// TwinCAT 3 PLC project TC
// ProgramVersion: 3.1.4022.3
// libraries:
//   Tc2_Standard, * (Beckhoff Automation GmbH)
//   Tc2_System, * (Beckhoff Automation GmbH)
//   Tc2_Utilities, * (Beckhoff Automation GmbH)
//   Tc3_EventLogger, * (Beckhoff Automation GmbH)
//   Tc3_HBI_Cylinder, * (BeckHoff SG)
//   Tc3_HBI_DataLogger, * (BeckHoff SG)
//   Tc3_HBI_System, * (BeckHoff)
//   Tc3_HBI_Utilities, * (BeckHoff SG)
//   Tc3_Module, * (Beckhoff Automation GmbH)
//   VisuDialogs, * (System)
//   VisuSymbols,3.5.10.0,System
// project tree:
//   DUTs/Actuator/ DUT_Cylinder.TcDUT, DUT_Switch.TcDUT, Enum_EPT.TcDUT, Enum_ModuleEnableState.TcDUT, Enum_Presence.TcDUT
//   DUTs/AIN/ DUT_AIN.TcDUT
//   DUTs/Enum/ E_AirValve.TcDUT, E_Cmd.TcTLEO, E_DBStnLED.TcDUT, E_FacilityState.TcDUT, E_LED.TcDUT, E_Pwr.TcDUT, E_Solenoid.TcDUT, E_TstPwrStep.TcDUT, E_BackdoorState_1.TcDUT, E_ModuleID_1.TcDUT, E_ProcessState.TcDUT, E_ProcessStep.TcDUT, E_SeqSts_1.TcDUT
//   DUTs/E_Alarm/ E_AlarmID.TcDUT, E_ColAlarm.TcDUT, E_DCFACAlarm.TcDUT, E_DSAlarm.TcDUT, E_TIIAlarm.TcDUT, ST_AlarmModules.TcDUT, ST_AlarmSubmodules.TcDUT, ST_AlarmTags.TcDUT
//   DUTs/Communication/ E_EventName.TcDUT, E_ModuleID.TcDUT, E_TaskName.TcDUT, ST_Command.TcDUT, ST_Event.TcDUT, ST_EventQueue.TcDUT, ST_TACommands.TcDUT, ST_TAEvents.TcDUT
//   DUTs/ E_BackdoorState.TcDUT, ST_StepMode.TcDUT, ST_DebugStation.TcDUT, ST_TCMultilevel.TcDUT, ST_TCShuttlePOC.TcDUT, ST_TCLevel.TcDUT
//   DUTs/HMI/ ST_BypassTII.TcDUT
//   DUTs/Logging/ F_Concat5.TcPOU
//   DUTs/ModuleState/EnableDisable/ E_State.TcDUT, ST_LPState.TcDUT, ST_LPTTS_State.TcDUT, ST_TCSubModuleState.TcDUT, ST_TCSiteState.TcDUT, ST_TTS_State.TcDUT
//   DUTs/ModuleState/EPT/ E_EPT.TcDUT, ST_LPTTS_EPT.TcDUT, ST_TCUEPT.TcDUT, ST_TCSubModuleEPT.TcDUT, ST_TC_EPT.TcDUT, ST_TTS_EPT.TcDUT
//   / GlobalTextList.TcGTLO, PlcTask.TcTTO, Visualization Manager.TcVMO (not stored)
//   GVLs/ AlarmTxtList.TcTLO, BDList.TcTLO, BtnTxtList.TcTLO, CmdTxtList.TcTLO, GVL_CONSTANTS.TcGVL, GVL_EAP.TcGVL, GVL_Motor.TcGVL, GVL_Process.TcGVL, GVL_SEN_SPEC.TcGVL, GVL_TA.TcGVL, GVL_TC.TcGVL, LevelTxtList.TcTLO
//   Image/ ImageCollection.TcIPO (not stored)
//   POUs/1%29 Main/ MAIN.TcPOU (not stored)
//   POUs/2%29 DFB/Actuator/ DFB_Cylinder.TcPOU (not stored)
//   POUs/2%29 DFB/ DFB_AIN.TcPOU (not stored), DFB_Second_Pulse.TcPOU (not stored), DFB_Switch.TcPOU (not stored)
//   POUs/2) DFB/Facility/ DFB_FacilityAlarmAnlg.TcPOU, DFB_FacilityAlarm.TcPOU, DFB_FacilityAlarm_1.TcPOU
//   POUs/2%29 DFB/Facility/ DFB_FacilityAlarmBool.TcPOU (not stored)
//   POUs/2%29 DFB/Word/ FC_BitToWord.TcPOU (not stored), FC_WordToBit.TcPOU (not stored)
//   POUs/3%29 FB/1%29 Common/EAP/ ST_DCEAP.TcDUT (not stored), ST_EAP.TcDUT (not stored), ST_TBOT_TC_EAP.TcDUT (not stored), ST_TBOT_TC_SubLevelEAP.TcDUT (not stored)
//   POUs/3%29 FB/1%29 Common/FB_Alarm/ FB_Alarm.TcPOU (not stored), FB_AlarmDelay.TcPOU (not stored), FB_Delay.TcPOU (not stored)
//   POUs/3%29 FB/1%29 Common/FB_CommonFunction/ FB_AnlgSIM.TcPOU (not stored), FB_Blink.TcPOU (not stored), F_ArrayInt.TcPOU (not stored), F_ArrayStr.TcPOU (not stored), F_Concat3.TcPOU (not stored), F_GetColumnID.TcPOU (not stored), F_GetModuleID.TcPOU (not stored), F_TAParamtoStr.TcPOU (not stored)
//   POUs/3%29 FB/1%29 Common/FB_EPT/ FB_DebugStationEPTUpdate.TcPOU (not stored), FB_TCMLevelEPTUpdate.TcPOU (not stored)
//   POUs/3%29 FB/1%29 Common/FB_Logging/ FB_AlarmMonitor.TcPOU (not stored), FB_SensorMonitor.TcPOU (not stored), F_AlarmLog.TcPOU (not stored), F_SensorLog.TcPOU (not stored), Logging.TcPOU (not stored)
//   POUs/3%29 FB/1%29 Common/FB_RemoteCmdAndEvent/ CmdAndEventProcess.TcPOU (not stored), FB_CmdAndEventUpdate.TcPOU (not stored), FB_DoorOpenClose.TcPOU (not stored), FB_TCUSafeState.TcPOU (not stored), FUN_CmdToEvent.TcPOU (not stored)
//   POUs/3%29 FB/2%29 TC/ ASSIGN_COLUMN.TcPOU (not stored), FB_UpdateStatus.TcPOU (not stored), PreInitialise.TcPOU (not stored)
//   POUs/3%29 FB/2%29 TC/FB_TCColumn/ FB_ColAlarm.TcPOU (not stored), FB_TCColumn.TcPOU (not stored), ST_TCColumn_BIO.TcDUT (not stored), ST_TCColumn_DIO.TcDUT (not stored), ST_TCColumn_VIO.TcDUT (not stored)
//   POUs/3%29 FB/2%29 TC/FB_TCMultiLevel/ FB_TCMLTesterPower_Process.TcPOU (not stored), FB_TCMultiLevelSeq.TcPOU (not stored), FB_TCMultiLevel_Process.TcPOU (not stored), FB_TIIAlarm.TcPOU (not stored), ST_TCMultiLevelSeqParam.TcDUT (not stored), ST_TCMultiLevel_BIO.TcDUT (not stored), ST_TCMultiLevel_DIO.TcDUT (not stored), ST_TCMultiLevel_VIO.TcDUT (not stored)
//   POUs/3%29 FB/2%29 TC/FB_TCShuttlePOC/ FB_TCShuttlePOCSeq.TcPOU (not stored), FB_TCShuttlePOC_Process.TcPOU (not stored), ST_TCSeqParam.TcDUT (not stored), ST_TCShuttlePOC_BIO.TcDUT (not stored), ST_TCShuttlePOC_DIO.TcDUT (not stored), ST_TCShuttlePOC_VIO.TcDUT (not stored)
//   POUs/3%29 FB/3%29 Debug Cart/FB_DebugStation/ FB_DBStnUpdateStatus.TcPOU (not stored), ANLG_TO_ABC.TcPOU (not stored), FB_DebugStationProcess.TcPOU (not stored), FB_DebugStationSeq.TcPOU (not stored), FB_TIIAlarmDbStn.TcPOU (not stored), ST_DebugStationSeqParam.TcDUT (not stored), ST_DebugStation_BIO.TcDUT (not stored), ST_DebugStation_DIO.TcDUT (not stored), ST_DebugStation_VIO.TcDUT (not stored), ST_SenSpec.TcDUT (not stored)
//   POUs/3) FB/2) TC/Testing/ CycleTest.TcPOU, EAPUpdate.TcPOU (not stored), FB_GUI_TEST.TcPOU, FB_GUI_TEST_SLTC.TcPOU, Testing.TcPOU, TestManually.TcPOU
//   POUs/3%29 FB/3%29 Debug Cart/Facility/ FB_Facility.TcPOU (not stored)
//   POUs/3%29 FB/3%29 Debug Cart/FB_DebugColumn/ FB_DebugColumn.TcPOU (not stored), ST_DebugColumnBIO.TcDUT (not stored), ST_DebugColumnDIO.TcDUT (not stored), ST_DebugColumnVIO.TcDUT (not stored)
//   POUs/3%29 FB/9%29 Unknown/ CheckBounds.TcPOU (not stored), CheckDivDInt.TcPOU (not stored), CheckDivLInt.TcPOU (not stored), CheckDivLReal.TcPOU (not stored) (excluded from build), CheckDivReal.TcPOU (not stored) (excluded from build), CheckLRangeSigned.TcPOU (not stored) (excluded from build), CheckLRangeUnsigned.TcPOU (not stored) (excluded from build), CheckPointer.TcPOU (not stored) (excluded from build), CheckRangeSigned.TcPOU (not stored) (excluded from build), CheckRangeUnsigned.TcPOU (not stored) (excluded from build)
//   POUs/3%29 FB/9%29 Unknown/FB_SLTC/ FB_Man_Stepping.TcPOU (not stored), FB_SLTC_EXTA.TcPOU (not stored), SLTC_EXTRA.TcPOU (not stored), ST_SLTC_EXTRA_BIO.TcDUT (not stored), ST_SLTC_EXTRA_DIO.TcDUT (not stored), ST_SLTC_EXTRA_VIO.TcDUT (not stored)
//   POUs/3%29 FB/9%29 Unknown/FB_TCLevel/DUTs/Enum/ E_SeqSts.TcDUT (not stored)
//   POUs/3%29 FB/9%29 Unknown/FB_TCLevel/ FB_TCLevelSeq.TcPOU (not stored), FB_TCLevel_Process.TcPOU (not stored), ST_TCLevel_BIO.TcDUT (not stored), ST_TCLevel_DIO.TcDUT (not stored), ST_TCLevel_VIO.TcDUT (not stored)
//   VISUs/ HMI_Alarm.TcVIS, HMI_DebugCell_Stack.TcVIS, HMI_DebugStation.TcVIS, HMI_FacilityAlarm_OFADewpoint.TcVIS, HMI_ManualCommand.TcVIS, HMI_OFA_Monitor.TcVIS, HMI_PCWBehaviour.TcVIS, HMI_PCW_Monitor.TcVIS, HMI_SenSimTest.TcVIS, HMI_All_Level.TcVIS, SLTC_Monitor.TcVIS
//   VISUs/Template/ AIN_Template.TcVIS, Cylinder_Template.TcVIS
// real-time tasks:
//   TASK PlcTask: cycle T#10ms, priority 6, ADS port 350
// I/O:
//   DEVICE Device 1 (EtherCAT), AmsNetId 192.168.1.4.2.1
//     Term 1 (EK1200) [EK1200-5000 EtherCAT Power supply (2A E-Bus)]
//       Term 2 (EL6070-0033) [EL6070-0033 1Ch. Licence key terminal, individual licences]
//       Term 3 (EK1122) [EK1122 2 port EtherCAT junction]
//         Term 4 (EK1101) [EK1101 EtherCAT Coupler (2A E-Bus, ID switch)]
//           Term 69 (EL1889) [EL1889 16Ch. Dig. Input 24V, 3ms, negative]
//           Term 70 (EL1889) [EL1889 16Ch. Dig. Input 24V, 3ms, negative]
//           Term 71 (EL1889) [EL1889 16Ch. Dig. Input 24V, 3ms, negative]
//           Term 72 (EL2889) [EL2889 16Ch. Dig. Output 24V, 0.5A, negative]
//           Term 73 (EL2889) [EL2889 16Ch. Dig. Output 24V, 0.5A, negative]
//           Term 15 (EL3104) [EL3104 4Ch. Ana. Input +/-10V Diff.] (disabled)
//           Term 16 (EL9011) [EL9011 End Terminal]
//         Term 10 (EK1101) [EK1101 EtherCAT Coupler (2A E-Bus, ID switch)]
//           Term 75 (EL1889) [EL1889 16Ch. Dig. Input 24V, 3ms, negative]
//           Term 76 (EL1889) [EL1889 16Ch. Dig. Input 24V, 3ms, negative]
//           Term 77 (EL1889) [EL1889 16Ch. Dig. Input 24V, 3ms, negative]
//           Term 78 (EL2889) [EL2889 16Ch. Dig. Output 24V, 0.5A, negative]
//           Term 79 (EL2889) [EL2889 16Ch. Dig. Output 24V, 0.5A, negative]
//           Term 17 (EL9011) [EL9011 End Terminal]
//   DEVICE Device 2 (EtherCAT Automation Protocol), AmsNetId 192.168.1.4.3.1
//     Box 5 (Publisher)
//     Box 6 (Subscriber)
// variable links:
//   TC/TC Instance <-> Device 1 (EtherCAT)/Term 1 (EK1200)/Term 3 (EK1122)/Term 10 (EK1101)/Term 75 (EL1889)
//     PlcTask Inputs/GVL_TC.arrTCMultiLevel[2].fbTCMultiLevelSeq.stMLDIO.ipAPPowerOn <-> Channel 2/Input
//     PlcTask Inputs/GVL_TC.arrTCMultiLevel[2].fbTCMultiLevelSeq.stMLDIO.ipAPPresentSensor <-> Channel 1/Input
//     PlcTask Inputs/GVL_TC.arrTCMultiLevel[2].fbTCMultiLevelSeq.stMLDIO.ipAPReady <-> Channel 3/Input
//     PlcTask Inputs/GVL_TC.arrTCMultiLevel[2].fbTCMultiLevelSeq.stMLDIO.ipCellFluidLeakage1 <-> Channel 10/Input
//     PlcTask Inputs/GVL_TC.arrTCMultiLevel[2].fbTCMultiLevelSeq.stMLDIO.ipCellFluidLeakage2 <-> Channel 11/Input
//     PlcTask Inputs/GVL_TC.arrTCMultiLevel[2].fbTCMultiLevelSeq.stMLDIO.ipCellGroundFault <-> Channel 12/Input
//     PlcTask Inputs/GVL_TC.arrTCMultiLevel[2].fbTCMultiLevelSeq.stMLDIO.ipHandlerSafeToEnterHwr <-> Channel 5/Input
//     PlcTask Inputs/GVL_TC.arrTCMultiLevel[2].fbTCMultiLevelSeq.stMLDIO.ipHandlerSafeToEnterPLC <-> Channel 4/Input
//     PlcTask Inputs/GVL_TC.arrTCMultiLevel[2].fbTCMultiLevelSeq.stMLDIO.ipSpare_1 <-> Channel 6/Input
//     PlcTask Inputs/GVL_TC.arrTCMultiLevel[2].fbTCMultiLevelSeq.stMLDIO.ipSpare_2 <-> Channel 7/Input
//     PlcTask Inputs/GVL_TC.arrTCMultiLevel[2].fbTCMultiLevelSeq.stMLDIO.ipSpare_3 <-> Channel 8/Input
//     PlcTask Inputs/GVL_TC.arrTCMultiLevel[2].fbTCMultiLevelSeq.stMLDIO.ipSpare_4 <-> Channel 9/Input
//     PlcTask Inputs/GVL_TC.arrTCMultiLevel[2].fbTCMultiLevelSeq.stMLDIO.ipSpare_5 <-> Channel 13/Input
//     PlcTask Inputs/GVL_TC.arrTCMultiLevel[2].fbTCMultiLevelSeq.stMLDIO.ipSpare_6 <-> Channel 14/Input
//     PlcTask Inputs/GVL_TC.arrTCMultiLevel[2].fbTCMultiLevelSeq.stMLDIO.ipSpare_7 <-> Channel 15/Input
//     PlcTask Inputs/GVL_TC.arrTCMultiLevel[2].fbTCMultiLevelSeq.stMLDIO.ipSpare_8 <-> Channel 16/Input
//   TC/TC Instance <-> Device 1 (EtherCAT)/Term 1 (EK1200)/Term 3 (EK1122)/Term 10 (EK1101)/Term 76 (EL1889)
//     PlcTask Inputs/GVL_TC.arrTCMultiLevel[2].fbTCMultiLevelSeq.stMLDIO.ipDrawerMaintenanceModeBtn <-> Channel 16/Input
//     PlcTask Inputs/GVL_TC.arrTCMultiLevel[2].fbTCMultiLevelSeq.stMLDIO.ipSpare_10 <-> Channel 5/Input
//     PlcTask Inputs/GVL_TC.arrTCMultiLevel[2].fbTCMultiLevelSeq.stMLDIO.ipSpare_9 <-> Channel 4/Input
//     PlcTask Inputs/GVL_TC.arrTCMultiLevel[2].fbTCMultiLevelSeq.stMLDIO.ipTCCellAbortFlowBtn <-> Channel 13/Input
//     PlcTask Inputs/GVL_TC.arrTCMultiLevel[2].fbTCMultiLevelSeq.stMLDIO.ipTCCellDoorClosed <-> Channel 10/Input
//     PlcTask Inputs/GVL_TC.arrTCMultiLevel[2].fbTCMultiLevelSeq.stMLDIO.ipTCCellDoorOpenCloseStatus <-> Channel 11/Input
//     PlcTask Inputs/GVL_TC.arrTCMultiLevel[2].fbTCMultiLevelSeq.stMLDIO.ipTCCellDoorOpenReqBtn <-> Channel 14/Input
//     PlcTask Inputs/GVL_TC.arrTCMultiLevel[2].fbTCMultiLevelSeq.stMLDIO.ipTCDrawerCylDownRS <-> Channel 9/Input
//     PlcTask Inputs/GVL_TC.arrTCMultiLevel[2].fbTCMultiLevelSeq.stMLDIO.ipTCDrawerCylExtendRS <-> Channel 6/Input
//     PlcTask Inputs/GVL_TC.arrTCMultiLevel[2].fbTCMultiLevelSeq.stMLDIO.ipTCDrawerCylRetractRS <-> Channel 7/Input
//     PlcTask Inputs/GVL_TC.arrTCMultiLevel[2].fbTCMultiLevelSeq.stMLDIO.ipTCDrawerCylUpRS <-> Channel 8/Input
//     PlcTask Inputs/GVL_TC.arrTCMultiLevel[2].fbTCMultiLevelSeq.stMLDIO.ipTIUPresent <-> Channel 15/Input
//     PlcTask Inputs/GVL_TC.arrTCMultiLevel[2].fbTCMultiLevelSeq.stMLDIO.ipTesterLatchesClosed <-> Channel 12/Input
//     PlcTask Inputs/GVL_TC.arrTCMultiLevel[2].fbTCMultiLevelSeq.stMLDIO.ipTesterPowerOn <-> Channel 2/Input
//     PlcTask Inputs/GVL_TC.arrTCMultiLevel[2].fbTCMultiLevelSeq.stMLDIO.ipTesterPresent <-> Channel 1/Input
//     PlcTask Inputs/GVL_TC.arrTCMultiLevel[2].fbTCMultiLevelSeq.stMLDIO.ipTesterReady <-> Channel 3/Input
//   TC/TC Instance <-> Device 1 (EtherCAT)/Term 1 (EK1200)/Term 3 (EK1122)/Term 10 (EK1101)/Term 77 (EL1889)
//     PlcTask Inputs/GVL_TC.arrTCMultiLevel[2].fbTCMultiLevelSeq.stMLDIO.ipTCCellTbotSideDoorLocked01 <-> Channel 3/Input
//     PlcTask Inputs/GVL_TC.arrTCMultiLevel[2].fbTCMultiLevelSeq.stMLDIO.ipTCCellTbotSideDoorLocked02 <-> Channel 4/Input
//     PlcTask Inputs/GVL_TC.arrTCMultiLevel[2].fbTCMultiLevelSeq.stMLDIO.ipTCCellTbotSideDoorOpenCloseStatus01 <-> Channel 1/Input
//     PlcTask Inputs/GVL_TC.arrTCMultiLevel[2].fbTCMultiLevelSeq.stMLDIO.ipTCCellTbotSideDoorOpenCloseStatus02 <-> Channel 2/Input
//   TC/TC Instance <-> Device 1 (EtherCAT)/Term 1 (EK1200)/Term 3 (EK1122)/Term 10 (EK1101)/Term 78 (EL2889)
//     PlcTask Outputs/GVL_TC.arrTCMultiLevel[2].fbTCMultiLevelSeq.stMLDIO.opAP240ACPwrEnable <-> Channel 1/Output
//     PlcTask Outputs/GVL_TC.arrTCMultiLevel[2].fbTCMultiLevelSeq.stMLDIO.opAPSafeToEngage <-> Channel 11/Output
//     PlcTask Outputs/GVL_TC.arrTCMultiLevel[2].fbTCMultiLevelSeq.stMLDIO.opAPTCCReset <-> Channel 12/Output
//     PlcTask Outputs/GVL_TC.arrTCMultiLevel[2].fbTCMultiLevelSeq.stMLDIO.opAlarmLED <-> Channel 6/Output
//     PlcTask Outputs/GVL_TC.arrTCMultiLevel[2].fbTCMultiLevelSeq.stMLDIO.opCellLTIMValve <-> Channel 16/Output
//     PlcTask Outputs/GVL_TC.arrTCMultiLevel[2].fbTCMultiLevelSeq.stMLDIO.opDoorOpenReqLED <-> Channel 5/Output
//     PlcTask Outputs/GVL_TC.arrTCMultiLevel[2].fbTCMultiLevelSeq.stMLDIO.opDrawerMaintenanceModeBtnLED <-> Channel 10/Output
//     PlcTask Outputs/GVL_TC.arrTCMultiLevel[2].fbTCMultiLevelSeq.stMLDIO.opSpare_1 <-> Channel 2/Output
//     PlcTask Outputs/GVL_TC.arrTCMultiLevel[2].fbTCMultiLevelSeq.stMLDIO.opSpare_2 <-> Channel 3/Output
//     PlcTask Outputs/GVL_TC.arrTCMultiLevel[2].fbTCMultiLevelSeq.stMLDIO.opSpare_3 <-> Channel 4/Output
//     PlcTask Outputs/GVL_TC.arrTCMultiLevel[2].fbTCMultiLevelSeq.stMLDIO.opSpare_6 <-> Channel 13/Output
//     PlcTask Outputs/GVL_TC.arrTCMultiLevel[2].fbTCMultiLevelSeq.stMLDIO.opSpare_7 <-> Channel 14/Output
//     PlcTask Outputs/GVL_TC.arrTCMultiLevel[2].fbTCMultiLevelSeq.stMLDIO.opSpare_8 <-> Channel 15/Output
//     PlcTask Outputs/GVL_TC.arrTCMultiLevel[2].fbTCMultiLevelSeq.stMLDIO.opTCCellAbortFlowBtnLED <-> Channel 9/Output
//   TC/TC Instance <-> Device 1 (EtherCAT)/Term 1 (EK1200)/Term 3 (EK1122)/Term 10 (EK1101)/Term 79 (EL2889)
//     PlcTask Outputs/GVL_TC.arrTCMultiLevel[2].fbTCMultiLevelSeq.stMLDIO.opAPAirSupplySol <-> Channel 11/Output
//     PlcTask Outputs/GVL_TC.arrTCMultiLevel[2].fbTCMultiLevelSeq.stMLDIO.opCell24VPowerEnable <-> Channel 13/Output
//     PlcTask Outputs/GVL_TC.arrTCMultiLevel[2].fbTCMultiLevelSeq.stMLDIO.opCellDoorClosed <-> Channel 16/Output
//     PlcTask Outputs/GVL_TC.arrTCMultiLevel[2].fbTCMultiLevelSeq.stMLDIO.opCellDrawerCylDown <-> Channel 4/Output
//     PlcTask Outputs/GVL_TC.arrTCMultiLevel[2].fbTCMultiLevelSeq.stMLDIO.opCellDrawerCylExtend <-> Channel 1/Output
//     PlcTask Outputs/GVL_TC.arrTCMultiLevel[2].fbTCMultiLevelSeq.stMLDIO.opCellDrawerCylRetract <-> Channel 2/Output
//     PlcTask Outputs/GVL_TC.arrTCMultiLevel[2].fbTCMultiLevelSeq.stMLDIO.opCellDrawerCylUp <-> Channel 3/Output
//     PlcTask Outputs/GVL_TC.arrTCMultiLevel[2].fbTCMultiLevelSeq.stMLDIO.opCellPCWValve <-> Channel 8/Output
//     PlcTask Outputs/GVL_TC.arrTCMultiLevel[2].fbTCMultiLevelSeq.stMLDIO.opCellTBOtSideDoorClosed1 <-> Channel 14/Output
//     PlcTask Outputs/GVL_TC.arrTCMultiLevel[2].fbTCMultiLevelSeq.stMLDIO.opCellTBOtSideDoorClosed2 <-> Channel 15/Output
//     PlcTask Outputs/GVL_TC.arrTCMultiLevel[2].fbTCMultiLevelSeq.stMLDIO.opSpare_10 <-> Channel 7/Output
//     PlcTask Outputs/GVL_TC.arrTCMultiLevel[2].fbTCMultiLevelSeq.stMLDIO.opSpare_9 <-> Channel 6/Output
//     PlcTask Outputs/GVL_TC.arrTCMultiLevel[2].fbTCMultiLevelSeq.stMLDIO.opTIUSktAirSol_1 <-> Channel 9/Output
//     PlcTask Outputs/GVL_TC.arrTCMultiLevel[2].fbTCMultiLevelSeq.stMLDIO.opTIUSktAirSol_2 <-> Channel 10/Output
//     PlcTask Outputs/GVL_TC.arrTCMultiLevel[2].fbTCMultiLevelSeq.stMLDIO.opTesterDrawerAirSupplySol <-> Channel 12/Output
//     PlcTask Outputs/GVL_TC.arrTCMultiLevel[2].fbTCMultiLevelSeq.stMLDIO.opTst240VACPwrEnable <-> Channel 5/Output
//   TC/TC Instance <-> Device 1 (EtherCAT)/Term 1 (EK1200)/Term 3 (EK1122)/Term 4 (EK1101)/Term 15 (EL3104)
//     PlcTask Inputs/GVL_TC.arrTCMultiLevel[1].fbTCMultiLevelSeq.stMLDIO.aiXAxis <-> AI Standard Channel 1/Value
//     PlcTask Inputs/GVL_TC.arrTCMultiLevel[1].fbTCMultiLevelSeq.stMLDIO.aiY1Axis <-> AI Standard Channel 4/Value
//     PlcTask Inputs/GVL_TC.arrTCMultiLevel[1].fbTCMultiLevelSeq.stMLDIO.aiYAxis <-> AI Standard Channel 2/Value
//     PlcTask Inputs/GVL_TC.arrTCMultiLevel[1].fbTCMultiLevelSeq.stMLDIO.aiZAxis <-> AI Standard Channel 3/Value
//   TC/TC Instance <-> Device 1 (EtherCAT)/Term 1 (EK1200)/Term 3 (EK1122)/Term 4 (EK1101)/Term 69 (EL1889)
//     PlcTask Inputs/GVL_TC.arrTCMultiLevel[1].fbTCMultiLevelSeq.stMLDIO.ipAPPowerOn <-> Channel 2/Input
//     PlcTask Inputs/GVL_TC.arrTCMultiLevel[1].fbTCMultiLevelSeq.stMLDIO.ipAPPresentSensor <-> Channel 1/Input
//     PlcTask Inputs/GVL_TC.arrTCMultiLevel[1].fbTCMultiLevelSeq.stMLDIO.ipAPReady <-> Channel 3/Input
//     PlcTask Inputs/GVL_TC.arrTCMultiLevel[1].fbTCMultiLevelSeq.stMLDIO.ipCellFluidLeakage1 <-> Channel 10/Input
//     PlcTask Inputs/GVL_TC.arrTCMultiLevel[1].fbTCMultiLevelSeq.stMLDIO.ipCellFluidLeakage2 <-> Channel 11/Input
//     PlcTask Inputs/GVL_TC.arrTCMultiLevel[1].fbTCMultiLevelSeq.stMLDIO.ipCellGroundFault <-> Channel 12/Input
//     PlcTask Inputs/GVL_TC.arrTCMultiLevel[1].fbTCMultiLevelSeq.stMLDIO.ipHandlerSafeToEnterHwr <-> Channel 5/Input
//     PlcTask Inputs/GVL_TC.arrTCMultiLevel[1].fbTCMultiLevelSeq.stMLDIO.ipHandlerSafeToEnterPLC <-> Channel 4/Input
//     PlcTask Inputs/GVL_TC.arrTCMultiLevel[1].fbTCMultiLevelSeq.stMLDIO.ipSpare_1 <-> Channel 6/Input
//     PlcTask Inputs/GVL_TC.arrTCMultiLevel[1].fbTCMultiLevelSeq.stMLDIO.ipSpare_2 <-> Channel 7/Input
//     PlcTask Inputs/GVL_TC.arrTCMultiLevel[1].fbTCMultiLevelSeq.stMLDIO.ipSpare_3 <-> Channel 8/Input
//     PlcTask Inputs/GVL_TC.arrTCMultiLevel[1].fbTCMultiLevelSeq.stMLDIO.ipSpare_4 <-> Channel 9/Input
//     PlcTask Inputs/GVL_TC.arrTCMultiLevel[1].fbTCMultiLevelSeq.stMLDIO.ipSpare_5 <-> Channel 13/Input
//     PlcTask Inputs/GVL_TC.arrTCMultiLevel[1].fbTCMultiLevelSeq.stMLDIO.ipSpare_6 <-> Channel 14/Input
//     PlcTask Inputs/GVL_TC.arrTCMultiLevel[1].fbTCMultiLevelSeq.stMLDIO.ipSpare_7 <-> Channel 15/Input
//     PlcTask Inputs/GVL_TC.arrTCMultiLevel[1].fbTCMultiLevelSeq.stMLDIO.ipSpare_8 <-> Channel 16/Input
//   TC/TC Instance <-> Device 1 (EtherCAT)/Term 1 (EK1200)/Term 3 (EK1122)/Term 4 (EK1101)/Term 70 (EL1889)
//     PlcTask Inputs/GVL_TC.arrTCMultiLevel[1].fbTCMultiLevelSeq.stMLDIO.ipDrawerMaintenanceModeBtn <-> Channel 16/Input
//     PlcTask Inputs/GVL_TC.arrTCMultiLevel[1].fbTCMultiLevelSeq.stMLDIO.ipSpare_10 <-> Channel 5/Input
//     PlcTask Inputs/GVL_TC.arrTCMultiLevel[1].fbTCMultiLevelSeq.stMLDIO.ipSpare_9 <-> Channel 4/Input
//     PlcTask Inputs/GVL_TC.arrTCMultiLevel[1].fbTCMultiLevelSeq.stMLDIO.ipTCCellAbortFlowBtn <-> Channel 13/Input
//     PlcTask Inputs/GVL_TC.arrTCMultiLevel[1].fbTCMultiLevelSeq.stMLDIO.ipTCCellDoorClosed <-> Channel 10/Input
//     PlcTask Inputs/GVL_TC.arrTCMultiLevel[1].fbTCMultiLevelSeq.stMLDIO.ipTCCellDoorOpenCloseStatus <-> Channel 11/Input
//     PlcTask Inputs/GVL_TC.arrTCMultiLevel[1].fbTCMultiLevelSeq.stMLDIO.ipTCCellDoorOpenReqBtn <-> Channel 14/Input
//     PlcTask Inputs/GVL_TC.arrTCMultiLevel[1].fbTCMultiLevelSeq.stMLDIO.ipTCDrawerCylDownRS <-> Channel 9/Input
//     PlcTask Inputs/GVL_TC.arrTCMultiLevel[1].fbTCMultiLevelSeq.stMLDIO.ipTCDrawerCylExtendRS <-> Channel 6/Input
//     PlcTask Inputs/GVL_TC.arrTCMultiLevel[1].fbTCMultiLevelSeq.stMLDIO.ipTCDrawerCylRetractRS <-> Channel 7/Input
//     PlcTask Inputs/GVL_TC.arrTCMultiLevel[1].fbTCMultiLevelSeq.stMLDIO.ipTCDrawerCylUpRS <-> Channel 8/Input
//     PlcTask Inputs/GVL_TC.arrTCMultiLevel[1].fbTCMultiLevelSeq.stMLDIO.ipTIUPresent <-> Channel 15/Input
//     PlcTask Inputs/GVL_TC.arrTCMultiLevel[1].fbTCMultiLevelSeq.stMLDIO.ipTesterLatchesClosed <-> Channel 12/Input
//     PlcTask Inputs/GVL_TC.arrTCMultiLevel[1].fbTCMultiLevelSeq.stMLDIO.ipTesterPowerOn <-> Channel 2/Input
//     PlcTask Inputs/GVL_TC.arrTCMultiLevel[1].fbTCMultiLevelSeq.stMLDIO.ipTesterPresent <-> Channel 1/Input
//     PlcTask Inputs/GVL_TC.arrTCMultiLevel[1].fbTCMultiLevelSeq.stMLDIO.ipTesterReady <-> Channel 3/Input
//   TC/TC Instance <-> Device 1 (EtherCAT)/Term 1 (EK1200)/Term 3 (EK1122)/Term 4 (EK1101)/Term 71 (EL1889)
//     PlcTask Inputs/GVL_TC.arrTCMultiLevel[1].fbTCMultiLevelSeq.stMLDIO.ipTCCellTbotSideDoorLocked01 <-> Channel 3/Input
//     PlcTask Inputs/GVL_TC.arrTCMultiLevel[1].fbTCMultiLevelSeq.stMLDIO.ipTCCellTbotSideDoorLocked02 <-> Channel 4/Input
//     PlcTask Inputs/GVL_TC.arrTCMultiLevel[1].fbTCMultiLevelSeq.stMLDIO.ipTCCellTbotSideDoorOpenCloseStatus01 <-> Channel 1/Input
//     PlcTask Inputs/GVL_TC.arrTCMultiLevel[1].fbTCMultiLevelSeq.stMLDIO.ipTCCellTbotSideDoorOpenCloseStatus02 <-> Channel 2/Input
//   TC/TC Instance <-> Device 1 (EtherCAT)/Term 1 (EK1200)/Term 3 (EK1122)/Term 4 (EK1101)/Term 72 (EL2889)
//     PlcTask Outputs/GVL_TC.arrTCMultiLevel[1].fbTCMultiLevelSeq.stMLDIO.opAP240ACPwrEnable <-> Channel 1/Output
//     PlcTask Outputs/GVL_TC.arrTCMultiLevel[1].fbTCMultiLevelSeq.stMLDIO.opAPSafeToEngage <-> Channel 11/Output
//     PlcTask Outputs/GVL_TC.arrTCMultiLevel[1].fbTCMultiLevelSeq.stMLDIO.opAPTCCReset <-> Channel 12/Output
//     PlcTask Outputs/GVL_TC.arrTCMultiLevel[1].fbTCMultiLevelSeq.stMLDIO.opAlarmLED <-> Channel 6/Output
//     PlcTask Outputs/GVL_TC.arrTCMultiLevel[1].fbTCMultiLevelSeq.stMLDIO.opCellLTIMValve <-> Channel 16/Output
//     PlcTask Outputs/GVL_TC.arrTCMultiLevel[1].fbTCMultiLevelSeq.stMLDIO.opDoorOpenReqLED <-> Channel 5/Output
//     PlcTask Outputs/GVL_TC.arrTCMultiLevel[1].fbTCMultiLevelSeq.stMLDIO.opDrawerMaintenanceModeBtnLED <-> Channel 10/Output
//     PlcTask Outputs/GVL_TC.arrTCMultiLevel[1].fbTCMultiLevelSeq.stMLDIO.opSpare_1 <-> Channel 2/Output
//     PlcTask Outputs/GVL_TC.arrTCMultiLevel[1].fbTCMultiLevelSeq.stMLDIO.opSpare_2 <-> Channel 3/Output
//     PlcTask Outputs/GVL_TC.arrTCMultiLevel[1].fbTCMultiLevelSeq.stMLDIO.opSpare_3 <-> Channel 4/Output
//     PlcTask Outputs/GVL_TC.arrTCMultiLevel[1].fbTCMultiLevelSeq.stMLDIO.opSpare_6 <-> Channel 13/Output
//     PlcTask Outputs/GVL_TC.arrTCMultiLevel[1].fbTCMultiLevelSeq.stMLDIO.opSpare_7 <-> Channel 14/Output
//     PlcTask Outputs/GVL_TC.arrTCMultiLevel[1].fbTCMultiLevelSeq.stMLDIO.opSpare_8 <-> Channel 15/Output
//     PlcTask Outputs/GVL_TC.arrTCMultiLevel[1].fbTCMultiLevelSeq.stMLDIO.opTCCellAbortFlowBtnLED <-> Channel 9/Output
//   TC/TC Instance <-> Device 1 (EtherCAT)/Term 1 (EK1200)/Term 3 (EK1122)/Term 4 (EK1101)/Term 73 (EL2889)
//     PlcTask Outputs/GVL_TC.arrTCMultiLevel[1].fbTCMultiLevelSeq.stMLDIO.opAPAirSupplySol <-> Channel 11/Output
//     PlcTask Outputs/GVL_TC.arrTCMultiLevel[1].fbTCMultiLevelSeq.stMLDIO.opCell24VPowerEnable <-> Channel 13/Output
//     PlcTask Outputs/GVL_TC.arrTCMultiLevel[1].fbTCMultiLevelSeq.stMLDIO.opCellDoorClosed <-> Channel 16/Output
//     PlcTask Outputs/GVL_TC.arrTCMultiLevel[1].fbTCMultiLevelSeq.stMLDIO.opCellDrawerCylDown <-> Channel 4/Output
//     PlcTask Outputs/GVL_TC.arrTCMultiLevel[1].fbTCMultiLevelSeq.stMLDIO.opCellDrawerCylExtend <-> Channel 1/Output
//     PlcTask Outputs/GVL_TC.arrTCMultiLevel[1].fbTCMultiLevelSeq.stMLDIO.opCellDrawerCylRetract <-> Channel 2/Output
//     PlcTask Outputs/GVL_TC.arrTCMultiLevel[1].fbTCMultiLevelSeq.stMLDIO.opCellDrawerCylUp <-> Channel 3/Output
//     PlcTask Outputs/GVL_TC.arrTCMultiLevel[1].fbTCMultiLevelSeq.stMLDIO.opCellPCWValve <-> Channel 8/Output
//     PlcTask Outputs/GVL_TC.arrTCMultiLevel[1].fbTCMultiLevelSeq.stMLDIO.opCellTBOtSideDoorClosed1 <-> Channel 14/Output
//     PlcTask Outputs/GVL_TC.arrTCMultiLevel[1].fbTCMultiLevelSeq.stMLDIO.opCellTBOtSideDoorClosed2 <-> Channel 15/Output
//     PlcTask Outputs/GVL_TC.arrTCMultiLevel[1].fbTCMultiLevelSeq.stMLDIO.opSpare_10 <-> Channel 7/Output
//     PlcTask Outputs/GVL_TC.arrTCMultiLevel[1].fbTCMultiLevelSeq.stMLDIO.opSpare_9 <-> Channel 6/Output
//     PlcTask Outputs/GVL_TC.arrTCMultiLevel[1].fbTCMultiLevelSeq.stMLDIO.opTIUSktAirSol_1 <-> Channel 9/Output
//     PlcTask Outputs/GVL_TC.arrTCMultiLevel[1].fbTCMultiLevelSeq.stMLDIO.opTIUSktAirSol_2 <-> Channel 10/Output
//     PlcTask Outputs/GVL_TC.arrTCMultiLevel[1].fbTCMultiLevelSeq.stMLDIO.opTesterDrawerAirSupplySol <-> Channel 12/Output
//     PlcTask Outputs/GVL_TC.arrTCMultiLevel[1].fbTCMultiLevelSeq.stMLDIO.opTst240VACPwrEnable <-> Channel 5/Output
//   TC/TC Instance <-> Device 2 (EtherCAT Automation Protocol)/Box 6 (Subscriber)
//     PlcTask Inputs/GVL_EAP.DS_Facility_eapShutOffAllACPower <-> eapShutOffAllAcPower/Inputs/eapShutOffAllACPower
//     PlcTask Inputs/GVL_TC.fbTCColumn.stTCColumnDIO.eapDColumnPCWLeakage <-> ColPCWLeakage/Inputs/VarData
//     PlcTask Inputs/GVL_TC.fbTCColumn.stTCColumnDIO.eapDColumnPCWLeakage2 <-> ColPCWLeakage2/Inputs/VarData
//     PlcTask Inputs/GVL_TC.fbTCColumn.stTCColumnDIO.eapDColumnPCWReturnLeakage <-> ColPCWReturnLeakage/Inputs/VarData
//     PlcTask Inputs/GVL_TC.fbTCColumn.stTCColumnDIO.eapDColumnPCWSupplyLeakage <-> ColPCWSupplyLeakage/Inputs/VarData

CONFIGURATION TC
    RESOURCE PLC ON TwinCAT3
        TASK PlcTask(INTERVAL := T#10ms, PRIORITY := 6);
        PROGRAM MAIN WITH PlcTask : MAIN;
        PROGRAM CycleTest WITH PlcTask : CycleTest;
    END_RESOURCE
END_CONFIGURATION

// ---- DUTs/Actuator/DUT_Cylinder.TcDUT
TYPE DUT_Cylinder :
STRUCT
	///////////////////////////////////////////////////////////////////////////////////////////////////////////////////////////////////////////
	// Settings
	///////////////////////////////////////////////////////////////////////////////////////////////////////////////////////////////////////////
	
	Simulate							: BOOL; // 0: Production mode, 1: Simulate mode
	Enable								: BOOL; // 0: Disable, 1: Enable
	Sim_Fail							: BOOL; // 0: Off, 1: Simulate Cylinder error
	SetOutput_Pulse						: BOOL; // 0: Command output will be keep updating, 1: Command output will be update once when there is state change
	Callibration_Mode					: BOOL; // 0: Ready for production, 1: Not ready for production
	
	
	///////////////////////////////////////////////////////////////////////////////////////////////////////////////////////////////////////////
	// Status
	///////////////////////////////////////////////////////////////////////////////////////////////////////////////////////////////////////////
	
	AutInp								: BOOL; // 0: Retract (Auto state), 1: Extend (Auto state)
	Failed								: BOOL; // 0: Cylinder OK, 1: Cylinder is failed to retract/extend*)
	Failed_To_Retract					: BOOL; // Failed to receive retract signal after travel time
	Failed_To_Extend					: BOOL; // Failed to receive extend signal after travel time
	
	Last_SD								: WORD; // Last Shut Down Error Code
	
	Status								: INT; // 1: Retracted, 2: Extended, 99: Failed
	
	Travel_Time							: UDINT	:= 5; // Time duration for DFB_Cylinder checking feedback input signal based on command output
	
	Message								: STRING; // Error Message
	
	EPT									: Enum_EPT; // 0: Blocked, 1: Idle, 2: Busy
	EnbState							: Enum_ModuleEnableState; // 0: Disabled, 1: Enabled
	Presence							: Enum_Presence; // 0: Non-Presence, 1: Presence
	
	
	///////////////////////////////////////////////////////////////////////////////////////////////////////////////////////////////////////////
	// Cylinder control & return
	///////////////////////////////////////////////////////////////////////////////////////////////////////////////////////////////////////////
	
	Reset								: BOOL; // 0: Idle, 1: Reset Motor
	
	CMD									: WORD	:= 4; // Command: 1: Retract, 2: Extend, 4: Auto
	
	
	///////////////////////////////////////////////////////////////////////////////////////////////////////////////////////////////////////////
	// Mapping
	///////////////////////////////////////////////////////////////////////////////////////////////////////////////////////////////////////////
	
	Extended							: BOOL;
	Retracted							: BOOL;
	Perm_BOOL							: ARRAY [1..16] OF BOOL;
	SD_BOOL								: ARRAY [1..16] OF BOOL;
	
	CylinderID							: STRING;
	Perm_STRING							: ARRAY [1..16] OF STRING;
	SD_STRING							: ARRAY [1..16] OF STRING;
END_STRUCT
END_TYPE

// ---- DUTs/Actuator/DUT_Switch.TcDUT
TYPE DUT_Switch :
STRUCT
	///////////////////////////////////////////////////////////////////////////////////////////////////////////////////////////////////////////
	// Settings
	///////////////////////////////////////////////////////////////////////////////////////////////////////////////////////////////////////////
	
	
	
	///////////////////////////////////////////////////////////////////////////////////////////////////////////////////////////////////////////
	// Status
	///////////////////////////////////////////////////////////////////////////////////////////////////////////////////////////////////////////
	
	
	
	///////////////////////////////////////////////////////////////////////////////////////////////////////////////////////////////////////////
	// Control & return
	///////////////////////////////////////////////////////////////////////////////////////////////////////////////////////////////////////////
	
	Q									: BOOL; 
	
	
	///////////////////////////////////////////////////////////////////////////////////////////////////////////////////////////////////////////
	// Mapping
	///////////////////////////////////////////////////////////////////////////////////////////////////////////////////////////////////////////
END_STRUCT
END_TYPE

// ---- DUTs/Actuator/Enum_EPT.TcDUT
{attribute 'qualified_only'}
{attribute 'strict'}
TYPE Enum_EPT :
(
	eBlocked := 0,
	eIdle,
	eBusy
);
END_TYPE

// ---- DUTs/Actuator/Enum_ModuleEnableState.TcDUT
{attribute 'qualified_only'}
{attribute 'strict'}
TYPE Enum_ModuleEnableState :
(
	eDisabled				 := 0,
	eEnabled
);
END_TYPE

// ---- DUTs/Actuator/Enum_Presence.TcDUT
{attribute 'qualified_only'}
{attribute 'strict'}
TYPE Enum_Presence :
(
	Non_presence := 0,				
	Presence
);
END_TYPE

// ---- DUTs/AIN/DUT_AIN.TcDUT
TYPE DUT_AIN :
STRUCT
	AIN_ID							: STRING; // AIN ID
	Simulate						: BOOL; // Simulation
	Healthy							: BOOL; // Healthy bit
	AHH_Enable						: BOOL; // Enable high high alarm
	AH_Enable						: BOOL; // Enable high alarm
	AL_Enable						: BOOL; // Enable low alarm
	ALL_Enable						: BOOL; // Enable low low alarm
	AHH								: BOOL; // High high alarm
	AH								: BOOL; // High alarm
	AL								: BOOL; // Low alarm
	ALL								: BOOL; // Low low alarm
	
	PV								: LREAL; // Process value
	AHH_SP							: LREAL; // High high alarm set point
	AH_SP							: LREAL; // High alarm set point
	AL_SP							: LREAL; // Low alarm set point
	ALL_SP							: LREAL; // Low low alarm set point
	DB								: LREAL; // Deadband
END_STRUCT
END_TYPE

// ---- DUTs/Enum/E_AirValve.TcDUT
{attribute 'qualified_only'}
{attribute 'strict'}
TYPE E_AirValve :
(
	UNKNOWN		:=0,
	TESTER	 	:=1,
	AP		 	:=2,
	TIU_SKT1 	:=3,
	TIU_SKT2 	:=4
);
END_TYPE

// ---- DUTs/Enum/E_Cmd.TcTLEO
{attribute 'qualified_only'}
{attribute 'strict'}
TYPE E_Cmd :
( 	
	INITIALISE:=0,
	AlarmReset,
	ColumnAlarmReset,
	TIUSlideIn,
	TIUSlideOut,
	TIUDrawerUp,
	TIUDrawerDown,
	TIUSlideOutRetry,
	TIUSlideOutCancel,
	DPSPowerON,
	DPSPowerOFF,
	DPSPowerAuto,
	AP240ACPowerON,
	AP240ACPowerOFF,
	APAirValveON,
	APAirValveOFF,
	TstAirValveON,
	TstAirValveOFF,
	CellDoorOpen,
	CellDoorClose,
	CancelBuffer,
	SetLEDON,
	SetLEDOFF, 
	SetLEDBlink,
	DCCellFrontDoorOpen,
	DCCellFrontDoorClose,
	TIUSocketAirOn_1,
	TIUSocketAirOn_2,
	TIUSocketAirOff_1,
	TIUSocketAirOff_2,
	EnableTester,
	DisableTester,
	EnableTCU,
	DisableTCU,
	EnableTII,
	DisableTII,
	SetTCUSafeState,
	SetSolenoidValvesON,
	SetSolenoidValvesOFF,
	Secondary24VPowerON,
	Secondary24VPowerOFF
);
END_TYPE

// ---- DUTs/Enum/E_DBStnLED.TcDUT
{attribute 'qualified_only'}
{attribute 'strict'}
TYPE E_DBStnLED :
(
	PurgeButton	:= 5
);
END_TYPE

// ---- DUTs/Enum/E_FacilityState.TcDUT
TYPE E_FacilityState :
(
	idle			:= 1,
	warningDelay,
	alarmDelay,
	warningDelayExpired,
	alarmDelayExpired,
	abortDelay,
	abortDelayExpired
);
END_TYPE

// ---- DUTs/Enum/E_LED.TcDUT
{attribute 'qualified_only'}
{attribute 'strict'}
TYPE E_LED :
(
	MaintenanceBtn := 0,
	AbortFlowBtn,
	DoorUnlockBtn,
	Aarm
);
END_TYPE

// ---- DUTs/Enum/E_Pwr.TcDUT
{attribute 'qualified_only'}
{attribute 'strict'}
TYPE E_Pwr :
(
	UNKNOWN:=0,
	ON,
	OFF,
	DONE
);
END_TYPE

// ---- DUTs/Enum/E_Solenoid.TcDUT
TYPE E_Solenoid :
(
	opDBStnPCWValve			:= 1,	//main pcw supply : OFF when perform purge
	opDBStnMainPCWReturn	:= 2,	//OFF when perform purge
	opDBStnPCWSupplyPurge	:= 3,	//OFF when perform purge
	opDBStnPCWAWN			:= 4,	//ON when perform purge
	opDBStnSupplyAirPurge	:= 5,	//ON when perform purge
	opDBStnLeakFlowPCWValve	:= 6,	
	opDBStnLowFlowPCWValve	:= 7
);
END_TYPE

// ---- DUTs/Enum/E_TstPwrStep.TcDUT
//{attribute 'qualified_only'}
//{attribute 'strict'}
TYPE E_TstPwrStep :
(
	INIT				,
	CheckCmd 			,
	SanityCheck		  	,	
	CheckCycPwr         ,
	ChkPwrOutputOn      ,
	OFF_PWR_FOR_CYC     ,
	WAIT_5              ,
	ON_PWR              ,
	WAIT_20             ,
	SetPwrOnTimeOutErr  ,
	ChkPwrOnFeedBack    ,
	ON_PCW              ,
	OFF_PWR_FOR_ERR     ,
	SEND_EVENT			,
	
	OFF_PWR				,
	OFF_PCW
);
END_TYPE

// ---- DUTs/E_Alarm/E_AlarmID.TcDUT
{attribute 'qualified_only'}
{attribute 'strict'}
TYPE E_AlarmID :
(

	DrawerExtendError 			:=31,	//31
	DrawerRetractError,					//32
	DrawerUpError,						//33
	DrawerDownError,					//34	
	TBotEAPNotSafeToMoveError,			//35
	TBotEAPAntiCollisionTriggered,		//36
	BothTIUExternRetractSignalDetected,	//37
	BothTIUUpDownSignalDetected,		//38
	APIsNotInUPPosition,				//39
	DoorCloseSignalNotDetected,			//40
	TBotSideDoorCloseSignalNotDetected	//41

);
END_TYPE

// ---- DUTs/E_Alarm/E_ColAlarm.TcDUT
{attribute 'qualified_only'}
{attribute 'strict'}
TYPE E_ColAlarm :
(
	ipColumnFluid_PCW_Leakage :=1,
    ipAllTCDrawerRetractedinCell,
	ipTbotDoorClosedSignal	
);
END_TYPE

// ---- DUTs/E_Alarm/E_DCFACAlarm.TcDUT
{attribute 'qualified_only'}
{attribute 'strict'}
//TYPE E_DCFACAlarm :
//(
//	ePCWSupplyHighTempWarning 		:=1,
//	e6BarLowOFAAirPressureWarning	,
//	e9BarLowOFAAirPressureWarning	,
//	eExcessiveHeatLoadIntoPCWWarning,
//	eCondensationWarning			,
//	eCriticalCondensationAlarm		,
//	eSystemPCWLeakageAlarm			,
//	eSystemPCWSupplyLeakageAlarm	,
//	eSystemPCWReturnLeakageAlarm
//);
//END_TYPE

TYPE E_DCFACAlarm :
(
	eSystemPCWLeakageAlarm				:= 1	,
	eSystemPCWSupplyLeakageAlarm     	:= 2    ,
	eSystemPCWReturnLeakageAlarm     	:= 3    ,
	eCriticalCondensationAlarm       	:= 4    ,
	e6BarLowOFAAirPressureAlarm			:= 5	,
	eSystemPCWLeakage2Alarm				:= 6	,
	ePCWSupplyHighTempWarning 			:= 11   ,
	e6BarLowOFAAirPressureWarning    	:= 12   ,
	e9BarLowOFAAirPressureWarning    	:= 13   ,
	eExcessiveHeatLoadIntoPCWWarning 	:= 14   ,
	eCondensationWarning             	:= 15   
);
END_TYPE

// ---- DUTs/E_Alarm/E_DSAlarm.TcDUT
{attribute 'qualified_only'}
{attribute 'strict'}
TYPE E_DSAlarm :
(
	eDBStnCellGroundFault := 1
);
END_TYPE

// ---- DUTs/E_Alarm/E_TIIAlarm.TcDUT
{attribute 'qualified_only'}
{attribute 'strict'}
TYPE E_TIIAlarm :
(
	ipAPPresentSensor		    		:= 1,
	ipAPPowerOn	 		    			,		//:=2
	ipAPReady				    		,		//:=3 
	ipAPDeactuatedPLC		    		,		//:=4
	ipAPDeactuatedHwr		    		,		//:=5
	ipCellFluidLeakage1		    		,		//:=6
	ipCellFluidLeakage2		  			,		//:=7
	ipCellGroundFault 		    		,		//:=8
	ipTesterPresent			    		,		//:=9
	ipTesterPowerOn			    		,		//:=10
	ipTesterReady			    		,		//:=11
	ipTCCellDoorClosed		    		,		//:=12
	ipTesterLatchesClosed	    		,		//:=13
	TBOT_TC_ACPower_Signal      		,		//:=14
	DS_Facility_EAP_ACPower_Signal		,		//:=15
	FrontDoorLockSignalNotDetected		,		//:=16
	ipTCDrawerExtendSignal				,		//:=17
	ipTCDrawerRetractSignal				,		//:=18
	ipTCDrawerUpSignal					,		//:=19
	ipTCDrawerDownSignal						//:=20
);
END_TYPE

// ---- DUTs/E_Alarm/ST_AlarmModules.TcDUT
TYPE ST_AlarmModules :
STRUCT
	Level:ARRAY[1..NO_OF_LEVEL] OF ST_AlarmTags;
	Common:ST_AlarmTags;
END_STRUCT
END_TYPE

// ---- DUTs/E_Alarm/ST_AlarmSubmodules.TcDUT
TYPE ST_AlarmSubmodules :
STRUCT
	AlarmSubmodule: ARRAY [1..30] OF ST_AlarmTags;
END_STRUCT
END_TYPE

// ---- DUTs/E_Alarm/ST_AlarmTags.TcDUT
TYPE ST_AlarmTags :
STRUCT
	AlarmID: ARRAY [1..NO_OF_ALARM_TAG] OF BOOL;
END_STRUCT
END_TYPE

// ---- DUTs/Communication/E_EventName.TcDUT
{attribute 'qualified_only'}
{attribute 'strict'}
TYPE E_EventName :
(
//(*
	//New
	EmptyEvent:=0,
	ValidateRecipeCompleted								:= 1	 ,
	ActivateRecipeCompleted                             := 2     ,
	ActivateRecipeFailed                                := 3     ,
	EnableModuleCompleted                               := 4     ,
	DisableModuleCompleted                              := 5     ,
	UpdateLCDCompleted                                  := 6     ,
	UpdateLCDFailed                                     := 7     ,
	GantryPickAndPlaceCompleted                         := 8     ,
	GantryPickAndPlaceFailed                            := 9     ,
	TBOTPickAndPlaceCompleted                           := 10    ,
	TBOTPickAndPlaceFailed                              := 11    ,
	SetLogVerbosityCompleted                            := 12    ,
	InitializeCompleted                                 := 13    ,
	InitializeFailed                                    := 14    ,
	ResumeCompleted                                     := 15    ,
	ResumeFailed                                        := 16    ,
	JogCompleted                                        := 17    ,
	JogFailed                                           := 18    ,
	AutoTeachCompleted                                  := 19    ,
	AutoTeachFailed                                     := 20    ,
	ApplyTeachDataCompleted                             := 21    ,
	ApplyTeachDataFailed                                := 22    ,
	AbortTeachCompleted                                 := 23    ,
	AbortTeachFailed                                    := 24    ,
	PauseCompleted                                      := 25    ,
	AlarmResetCompleted                                 := 26    ,
	AlarmResetFailed                                    := 27    ,
	AlarmCleared                                        := 28    ,
	WriteRFIDDataCompleted                              := 29    ,
	WriteRFIDDataFailed                                 := 30    ,
	MoveGantryCompleted                                 := 31    ,
	MoveGantryFailed                                    := 32    ,
	MoveTBOTCompleted                                   := 33    ,
	MoveTBOTFailed                                      := 34    ,
	DoorOpenCompleted                                   := 35    ,
	DoorOpenFailed                                      := 36    ,
	DoorCloseCompleted                                  := 37    ,
	DoorCloseFailed                                     := 38    ,
	CancelCompleted                                     := 39    ,
	MoveTBOTRetryCompleted                              := 40    ,
	MoveTBOTRetryFailed                                 := 41    ,
	MoveTBOTCancelCompleted                             := 42    ,
	MoveTBOTCancelFailed                                := 43    ,
	TBOTPickAndPlaceRetryCompleted                      := 44    ,
	TBOTPickAndPlaceRetryFailed                         := 45    ,
	TBOTPickAndPlaceCancelCompleted                     := 46    ,
	TBOTPickAndPlaceCancelFailed                        := 47    ,
	MoveGantryRetryCompleted                            := 48    ,
	MoveGantryRetryFailed                               := 49    ,
	MoveGantryCancelCompleted                           := 50    ,
	MoveGantryCancelFailed                              := 51    ,
	GantryPickAndPlaceRetryCompleted                    := 52    ,
	GantryPickAndPlaceRetryFailed                       := 53    ,
	GantryPickAndPlaceCancelCompleted                   := 54    ,
	GantryPickAndPlaceCancelFailed                      := 55    ,
	SingulateTrayStackerRetryCompleted                  := 56    ,
	SingulateTrayStackerRetryFailed                     := 57    ,
	SingulateTrayStackerCancelCompleted                 := 58    ,
	SingulateTrayStackerCancelFailed                    := 59    ,
	SingulateTrayStackerHalfRetryCompleted              := 60    ,
	SingulateTrayStackerHalfRetryFailed                 := 61    ,
	SingulateTrayStackerHalfCancelCompleted             := 62    ,
	SingulateTrayStackerHalfCancelFailed                := 63    ,
	SingulateTrayStackerRemainingRetryCompleted         := 64    ,
	SingulateTrayStackerRemainingRetryFailed            := 65    ,
	SingulateTrayStackerRemainingCancelCompleted        := 66    ,
	SingulateTrayStackerRemainingCancelFailed           := 67    ,
	StackUpTrayStackerRetryCompleted                    := 68    ,
	StackUpTrayStackerRetryFailed                       := 69    ,
	StackUpTrayStackerCancelCompleted                   := 70    ,
	StackUpTrayStackerCancelFailed                      := 71    ,
	MoveConveyorForwardRetryCompleted                   := 72    ,
	MoveConveyorForwardRetryFailed                      := 73    ,
	MoveConveyorForwardCancelCompleted                  := 74    ,
	MoveConveyorForwardCancelFailed                     := 75    ,
	MoveConveyorBackwardRetryCompleted                  := 76    ,
	MoveConveyorBackwardRetryFailed                     := 77    ,
	MoveConveyorBackwardCancelCompleted                 := 78    ,
	MoveConveyorBackwardCancelFailed                    := 79    ,
	MoveVisionShuttleRetryCompleted                     := 80    ,
	MoveVisionShuttleRetryFailed                        := 81    ,
	MoveVisionShuttleCancelCompleted                    := 82    ,
	MoveVisionShuttleCancelFailed                       := 83    ,
	MoveUPortShuttleRetryCompleted                      := 84    ,
	MoveUPortShuttleRetryFailed                         := 85    ,
	MoveUPortShuttleCancelCompleted                     := 86    ,
	MoveUPortShuttleCancelFailed                        := 87    ,
	MoveFlyoverShuttleRetryCompleted                    := 88    ,
	MoveFlyoverShuttleRetryFailed                       := 89    ,
	MoveFlyoverShuttleCancelCompleted                   := 90    ,
	MoveFlyoverShuttleCancelFailed                      := 91    ,
	MoveTrayScanShuttleRetryCompleted                   := 92    ,
	MoveTrayScanShuttleRetryFailed                      := 93    ,
	MoveTrayScanShuttleCancelCompleted                  := 94    ,
	MoveTrayScanShuttleCancelFailed                     := 95    ,
	MoveTrayScanShuttleLifterRetryCompleted             := 96    ,
	MoveTrayScanShuttleLifterRetryFailed                := 97    ,
	MoveTrayScanShuttleLifterCancelCompleted            := 98    ,
	MoveTrayScanShuttleLifterCancelFailed               := 99    ,
	DPSPowerCompleted                                   := 100   ,
	DPSPowerFailed                                      := 101   ,
	ReadRFIDCompleted                                   := 102   ,
	ReadRFIDFailed                                      := 103   ,
	UnitPresentCheckFailed                              := 104   ,
	UnitPresentCheckCompleted                           := 105   ,
	TrayClampCompleted                                  := 106   ,
	TrayClampFailed                                     := 107   ,
	ChangeStackCountCompleted                           := 108   ,
	ChangeStackCountFailed                              := 109   ,
	BypassVisionCompleted                               := 110   ,
	PNBDoorUnlockRequest                                := 111   ,
	ButtonDoorLockCompleted                             := 112   ,
	PNBDoorLockRequest                                  := 113   ,
	CalibrationOffsetResult                             := 114   ,
	DoorRecoveryStarted                                 := 115   ,
	DoorRecoveryCompleted                               := 116   ,
	DoorRecoveryFailed                                  := 117   ,
	TCCSessionRequestCompleted                          := 118   ,
	TCCSessionRequestFailed                             := 119   ,
	TIUSlideOutCompleted                                := 120   ,
	TIUSlideOutFailed                                   := 121   ,
	PrecisorSlideOutCompleted                           := 122   ,
	PrecisorSlideOutFailed                              := 123   ,
	SingulateTrayStackerCompleted                       := 124   ,
	SingulateTrayStackerFailed                          := 125   ,
	SingulateTrayStackerHalfCompleted                   := 126   ,
	SingulateTrayStackerHalfFailed                      := 127   ,
	SingulateTrayStackerRemainingCompleted              := 128   ,
	SingulateTrayStackerRemainingFailed                 := 129   ,
	StackUpTrayStackerCompleted                         := 130   ,
	StackUpTrayStackerFailed                            := 131   ,
	StopperUpCompleted                                  := 132   ,
	StopperUpFailed                                     := 133   ,
	MoveConveyorForwardCompleted                        := 134   ,
	MoveConveyorForwardFailed                           := 135   ,
	MoveConveyorBackwardCompleted                       := 136   ,
	MoveConveyorBackwardFailed                          := 137   ,
	MoveVisionShuttleCompleted                          := 138   ,
	MoveVisionShuttleFailed                             := 139   ,
	MoveUPortShuttleCompleted                           := 140   ,
	MoveUPortShuttleFailed                              := 141   ,
	UPortShuttleReadyCompleted                          := 142   ,
	UPortShuttleReadyFailed                             := 143   ,
	MoveFlyoverShuttleCompleted                         := 144   ,
	MoveFlyoverShuttleFailed                            := 145   ,
	FlyoverShuttlePickCompleted                         := 146   ,
	FlyoverShuttlePickFailed                            := 147   ,
	FlyoverShuttlePlaceCompleted                        := 148   ,
	FlyoverShuttlePlaceFailed                           := 149   ,
	MoveTrayScanShuttleCompleted                        := 150   ,
	MoveTrayScanShuttleFailed                           := 151   ,
	MoveTrayScanShuttleLifterCompleted                  := 152   ,
	MoveTrayScanShuttleLifterFailed                     := 153   ,
	EportLatchCompleted                                 := 154   ,
	EportLatchFailed                                    := 155   ,
	TrayClearedSafetySensorCompleted                    := 156   ,
	TIUSlideOutRetryCompleted                           := 157   ,
	TIUSlideOutRetryFailed                              := 158   ,
	TIUSlideOutCancelCompleted                          := 159   ,
	TIUSlideOutCancelFailed                             := 160   ,
	MoveTTSShuttleCompleted                             := 161   ,
	MoveTTSShuttleFailed                                := 162   ,
	MoveTTSShuttleRetryCompleted                        := 163   ,
	MoveTTSShuttleRetryFailed                           := 164   ,
	MoveTTSShuttleCancelCompleted                       := 165   ,
	MoveTTSShuttleCancelFailed                          := 166   ,
	SingulateTrayLatchRemainingCompleted                := 167   ,
	SingulateTrayLatchRemainingFailed                   := 168   ,
	SingulateTrayLatchRemainingRetryCompleted           := 169   ,
	SingulateTrayLatchRemainingRetryFailed              := 170   ,
	SingulateTrayLatchRemainingCancelCompleted          := 171   ,
	SingulateTrayLatchRemainingCancelFailed             := 172   ,
	SingulateTrayLatchCompleted                         := 173   ,
	SingulateTrayLatchFailed                            := 174   ,
	SingulateTrayLatchRetryCompleted                    := 175   ,
	SingulateTrayLatchRetryFailed                       := 176   ,
	SingulateTrayLatchCancelCompleted                   := 177   ,
	SingulateTrayLatchCancelFailed                      := 178   ,
	StackUpTrayLatchCompleted                           := 179   ,
	StackUpTrayLatchFailed                              := 180   ,
	StackUpTrayLatchRetryCompleted                      := 181   ,
	StackUpTrayLatchRetryFailed                         := 182   ,
	StackUpTrayLatchCancelCompleted                     := 183   ,
	StackUpTrayLatchCancelFailed                        := 184   ,
	StackerTeachResult                                  := 185   ,
	UserButtonPressCompleted                            := 186   ,
	SingulateCylinderTrayCompleted                      := 187   ,
	SingulateCylinderTrayFailed                         := 188   ,
	SingulateCylinderTrayRetryCompleted                 := 189   ,
	SingulateCylinderTrayRetryFailed                    := 190   ,
	SingulateCylinderTrayCancelCompleted                := 191   ,
	SingulateCylinderTrayCancelFailed                   := 192   ,
	StackUpCylinderTrayCompleted                        := 193   ,
	StackUpCylinderTrayFailed                           := 194   ,
	StackUpCylinderTrayRetryCompleted                   := 195   ,
	StackUpCylinderTrayRetryFailed                      := 196   ,
	StackUpCylinderTrayCancelCompleted                  := 197   ,
	StackUpCylinderTrayCancelFailed                     := 198   ,
	SetUportBlinkRateCompleted                          := 199   ,
	SetUportBlinkRateFailed                             := 200   ,
	DrawerUpCompleted                                   := 201   ,
	DrawerUpFailed                                      := 202   ,
	AP240ACPwrCompleted                                 := 203   ,
	AP240ACPwrFailed                                    := 204   ,
	TesterAirValveCompleted                             := 205   ,
	TesterAirValveFailed                                := 206   ,
	APAirValveCompleted                                 := 207   ,
	APAirValveFailed                                    := 208   ,
	ManualButtonPressCompleted                          := 209   ,
	MoveToPosition 										:= 210	 ,
	LaneStackerResult 									:= 211	 ,
	SetBlinkRateCompleted 								:= 212	 ,
	TIUSocketCoolingAirCompleted 						:= 213	 ,
	SetSolenoidValvesCompleted							:= 263	 ,
	SetSolenoidValvesFailed								:= 264	 ,
	DewPointAbortInProgress 							:= 265	 ,
	SixbarOFAAbortInProgress							:= 266	 ,
	Secondary24VPowerCompleted							:= 271	 ,
	Secondary24VPowerFailed								:= 272

//*)       
                                                                                                                
(*   
	//Old                                                          
	EmptyEvent :=0,                                                
	ValidateRecipeCompleted :=1,                                   
	ActivateRecipeCompleted :=2,                                   
	ActivateRecipeFailed :=3,                                      
	EnableModuleCompleted :=4,                                     
	DisableModuleCompleted :=5,                                    
	UpdateLCDCompleted :=6,                                        
	UpdateLCDFailed :=7,                                           
	GantryPickAndPlaceCompleted :=8,                               
	GantryPickAndPlaceFailed :=9,                                  
	TBOTPickAndPlaceCompleted :=10,                                
	TBOTPickAndPlaceFailed :=11,                                   
	SetLogVerbosityCompleted :=12,                                 
	InitializeCompleted :=13,                                      
	InitializeFailed :=14,                                         
	ResumeCompleted :=15,                                          
	ResumeFailed :=16,                                             
	JogCompleted :=17,                                             
	JogFailed :=18,                                                
	AutoTeachCompleted :=19,                                       
	AutoTeachFailed :=20,                                          
	ApplyTeachDataCompleted :=21,                                  
	ApplyTeachDataFailed :=22,                                     
	AbortTeachCompleted :=23,
	AbortTeachFailed :=24,
	PauseCompleted :=25,
	AlarmResetCompleted :=26,
	AlarmResetFailed :=27,
	AlarmCleared :=28,
	WriteRFIDDataCompleted :=29,
	WriteRFIDDataFailed :=30,
	MoveGantryCompleted :=31,
	MoveGantryFailed :=32,
	MoveTBOTCompleted :=33,
	MoveTBOTFailed :=34,
	DoorOpenCompleted :=35,
	DoorOpenFailed :=36,
	DoorCloseCompleted :=37,
	DoorCloseFailed :=38,
	CancelCompleted :=39,
	MoveTBOTRetryCompleted :=40,
	MoveTBOTRetryFailed :=41,
	MoveTBOTCancelCompleted :=42,
	MoveTBOTCancelFailed :=43,
	TBOTPickAndPlaceRetryCompleted :=44,
	TBOTPickAndPlaceRetryFailed :=45,
	TBOTPickAndPlaceCancelCompleted :=46,
	TBOTPickAndPlaceCancelFailed :=47,
	MoveGantryRetryCompleted :=48,
	MoveGantryRetryFailed :=49,
	MoveGantryCancelCompleted :=50,
	MoveGantryCancelFailed :=51,
	GantryPickAndPlaceRetryCompleted :=52,
	GantryPickAndPlaceRetryFailed :=53,
	GantryPickAndPlaceCancelCompleted :=54,
	GantryPickAndPlaceCancelFailed :=55,
	SingulateTrayStackerRetryCompleted :=56,
	SingulateTrayStackerRetryFailed :=57,
	SingulateTrayStackerCancelCompleted :=58,
	SingulateTrayStackerCancelFailed :=59,
	SingulateTrayStackerHalfRetryCompleted :=60,
	SingulateTrayStackerHalfRetryFailed :=61,
	SingulateTrayStackerHalfCancelCompleted :=62,
	SingulateTrayStackerHalfCancelFailed :=63,
	SingulateTrayStackerRemainingRetryCompleted :=64,
	SingulateTrayStackerRemainingRetryFailed :=65,
	SingulateTrayStackerRemainingCancelCompleted :=66,
	SingulateTrayStackerRemainingCancelFailed :=67,
	StackUpTrayStackerRetryCompleted :=68,
	StackUpTrayStackerRetryFailed :=69,
	StackUpTrayStackerCancelCompleted :=70,
	StackUpTrayStackerCancelFailed :=71,
	MoveConveyorForwardRetryCompleted :=72,
	MoveConveyorForwardRetryFailed :=73,
	MoveConveyorForwardCancelCompleted :=74,
	MoveConveyorForwardCancelFailed :=75,
	MoveConveyorBackwardRetryCompleted :=76,
	MoveConveyorBackwardRetryFailed :=77,
	MoveConveyorBackwardCancelCompleted :=78,
	MoveConveyorBackwardCancelFailed :=79,
	MoveVisionShuttleRetryCompleted :=80,
	MoveVisionShuttleRetryFailed :=81,
	MoveVisionShuttleCancelCompleted :=82,
	MoveVisionShuttleCancelFailed :=83,
	MoveUPortShuttleRetryCompleted :=84,
	MoveUPortShuttleRetryFailed :=85,
	MoveUPortShuttleCancelCompleted :=86,
	MoveUPortShuttleCancelFailed :=87,
	MoveFlyoverShuttleRetryCompleted :=88,
	MoveFlyoverShuttleRetryFailed :=89,
	MoveFlyoverShuttleCancelCompleted :=90,
	MoveFlyoverShuttleCancelFailed :=91,
	MoveTrayScanShuttleRetryCompleted :=92,
	MoveTrayScanShuttleRetryFailed :=93,
	MoveTrayScanShuttleCancelCompleted :=94,
	MoveTrayScanShuttleCancelFailed :=95,
	MoveTrayScanShuttleLifterRetryCompleted :=96,
	MoveTrayScanShuttleLifterRetryFailed :=97,
	MoveTrayScanShuttleLifterCancelCompleted :=98,
	MoveTrayScanShuttleLifterCancelFailed :=99,
	DPSPowerCompleted :=100,
	DPSPowerFailed :=101,
	ReadIDCompleted :=102,
	ReadIDFailed :=103,
	UnitPresentCheckFailed :=104,
	UnitPresentCheckCompleted :=105,
	TrayClampCompleted :=106,
	TrayClampFailed :=107,
	ChangeStackCountCompleted :=108,
	ChangeStackCountFailed :=109,
	BypassVisionCompleted :=110,
	PNBDoorUnlockRequest :=111,
	ButtonDoorLockCompleted :=112,
	PNBDoorLockRequest :=113,
	CalibrationOffsetResult :=114,
	DoorRecoveryStarted :=115,
	DoorRecoveryCompleted :=116,
	DoorRecoveryFailed :=117,
	TCCSessionRequestCompleted :=118,
	TCCSessionRequestFailed :=119,
	TIUSlideOutCompleted :=120,
	TIUSlideOutFailed :=121,
	PrecisorSlideOutCompleted :=122,
	PrecisorSlideOutFailed :=123,
	SingulateTrayStackerCompleted :=124,
	SingulateTrayStackerFailed :=125,
	SingulateTrayStackerHalfCompleted :=126,
	SingulateTrayStackerHalfFailed :=127,
	SingulateTrayStackerRemainingCompleted :=128,
	SingulateTrayStackerRemainingFailed :=129,
	StackUpTrayStackerCompleted :=130,
	StackUpTrayStackerFailed :=131,
	StopperUpCompleted :=132,
	StopperUpFailed :=133,
	MoveConveyorForwardCompleted :=134,
	MoveConveyorForwardFailed :=135,
	MoveConveyorBackwardCompleted :=136,
	MoveConveyorBackwardFailed :=137,
	MoveVisionShuttleCompleted :=138,
	MoveVisionShuttleFailed :=139,
	MoveUPortShuttleCompleted :=140,
	MoveUPortShuttleFailed :=141,
	UPortShuttleReadyCompleted :=142,
	UPortShuttleReadyFailed :=143,
	MoveFlyoverShuttleCompleted :=144,
	MoveFlyoverShuttleFailed :=145,
	FlyoverShuttlePickCompleted :=146,
	FlyoverShuttlePickFailed :=147,
	FlyoverShuttlePlaceCompleted :=148,
	FlyoverShuttlePlaceFailed :=149,
	MoveTrayScanShuttleCompleted :=150,
	MoveTrayScanShuttleFailed :=151,
	MoveTrayScanShuttleLifterCompleted :=152,
	MoveTrayScanShuttleLifterFailed :=153,
	EportLatchCompleted :=154,
	EportLatchFailed :=155,
	TrayClearedSafetySensorCompleted :=156,
	TIUSlideOutRetryCompleted :=157,
	TIUSlideOutRetryFailed :=158,
	TIUSlideOutCancelCompleted :=159,
	TIUSlideOutCancelFailed :=160,
	MoveTTSShuttleCompleted :=161,
	MoveTTSShuttleFailed :=162,
	MoveTTSShuttleRetryCompleted :=163,
	MoveTTSShuttleRetryFailed :=164,
	MoveTTSShuttleCancelCompleted :=165,
	MoveTTSShuttleCancelFailed :=166,
	SingulateTrayLatchRemainingCompleted :=167,
	SingulateTrayLatchRemainingFailed :=168,
	SingulateTrayLatchRemainingRetryCompleted :=169,
	SingulateTrayLatchRemainingRetryFailed :=170,
	SingulateTrayLatchRemainingCancelCompleted :=171,
	SingulateTrayLatchRemainingCancelFailed :=172,
	SingulateTrayLatchCompleted :=173,
	SingulateTrayLatchFailed :=174,
	SingulateTrayLatchRetryCompleted :=175,
	SingulateTrayLatchRetryFailed :=176,
	SingulateTrayLatchCancelCompleted :=177,
	SingulateTrayLatchCancelFailed :=178,
	StackUpTrayLatchCompleted :=179,
	StackUpTrayLatchFailed :=180,
	StackUpTrayLatchRetryCompleted :=181,
	StackUpTrayLatchRetryFailed :=182,
	StackUpTrayLatchCancelCompleted :=183,
	StackUpTrayLatchCancelFailed :=184,
	StackerTeachResult :=185,
	UserButtonPressCompleted :=186,
	SingulateCylinderTrayCompleted :=187,
	SingulateCylinderTrayFailed :=188,
	SingulateCylinderTrayRetryCompleted :=189,
	SingulateCylinderTrayRetryFailed :=190,
	SingulateCylinderTrayCancelCompleted :=191,
	SingulateCylinderTrayCancelFailed :=192,
	StackUpCylinderTrayCompleted :=193,
	StackUpCylinderTrayFailed :=194,
	StackUpCylinderTrayRetryCompleted :=195,
	StackUpCylinderTrayRetryFailed :=196,
	StackUpCylinderTrayCancelCompleted :=197,
	StackUpCylinderTrayCancelFailed :=198,
	
	//joanne
	SetUportBlinkRateCompleted :=199,
	SetUportBlinkRateFailed :=200,
	//joanne
	(*SingulateCylinderTrayCompleted :=185,
	SingulateCylinderTrayFailed :=186,
	StackupCylinderTrayCompleted :=187,
	StackupCylinderTrayFailed :=188,
	
	SingulateCylinderTrayRetryCompleted :=189,
	SingulateCylinderTrayRetryFailed :=190,
	StackupCylinderTrayRetryCompleted :=191,
	StackupCylinderTrayRetryFailed :=192,
	SetUportBlinkRateCompleted :=193,
	SetUportBlinkRateFailed :=194,
	UserButtonPressCompleted :=195*)
	//StackerTeachResult (Depreceted?) ::=185
	
	(*AlarmTriggered :=161, //joanne new add
	CancelFailed :=162 //joanne new add
	//StackerTeachResult (Depreceted?) :=161,*)
	ManualButtonPressedCompleted:=700,
	DrawerUpCompleted :=701,
	DrawerUpFailed :=702,
	AP240ACPwrCompleted :=703,
	AP240ACPwrFailed :=704,
	TesterAirValveCompleted:=705,
	TesterAirValveFailed:=706,
	APAirValveCompleted:=707,
	APAirValveFailed:=708
*)
);

END_TYPE

// ---- DUTs/Communication/E_ModuleID.TcDUT
{attribute 'qualified_only'}
{attribute 'strict'}
TYPE E_ModuleID :
(


